FUNCTION_BLOCK fbPiston EXTENDS TcoCore.TcoSequencer

METHOD PROTECTED Main : BOOL


IF Step(10,
TRUE,
'_moveHomeTask') THEN
//-------------------------------------------------------
	IF(_moveHomeTask.Invoke().Done)THEN
		StepCompleteWhen(TRUE);
	END_IF;
//-------------------------------------------------------
END_IF;

IF Step(20,
TRUE,
'_moveWorkTask') THEN
//-------------------------------------------------------
	IF(_moveWorkTask.Invoke().Done)THEN
		StepCompleteWhen(TRUE);
	END_IF;
//-------------------------------------------------------
END_IF;

IF Step(30,
TRUE,
'_moveHomeToggleTask') THEN
//-------------------------------------------------------
	IF(_moveHomeToggleTask.Toggle())THEN
		StepCompleteWhen(TRUE);
	END_IF;
//-------------------------------------------------------
END_IF;

IF Step(40,
TRUE,
'_moveHomeToggleTask') THEN
//-------------------------------------------------------
	IF(_moveHomeToggleTask.Toggle())THEN
		StepCompleteWhen(TRUE);
	END_IF;
//-------------------------------------------------------
END_IF;

IF Step(50,
TRUE,
'_moveHomeMomentaryTask') THEN
//-------------------------------------------------------
	IF(_moveHomeMomentaryTask.On())THEN
		StepCompleteWhen(TRUE);
	END_IF;
//-------------------------------------------------------
END_IF;

IF Step(60,
TRUE,
'_moveHomeMomentaryTask') THEN
//-------------------------------------------------------
	IF(_moveHomeMomentaryTask.Off())THEN
		StepCompleteWhen(TRUE);
	END_IF;
//-------------------------------------------------------
END_IF;
END_METHOD

END_FUNCTION_BLOCK

(* stored: Version 1.1.0.1, ProductVersion 3.1.4024.9
   POU fbPiston: Id {41ce95b1-694a-4bd3-b773-5382b98402d8}, SpecialFunc None
   Method Main: Id {c86ecde6-1911-404c-86d2-9ddbfc0b3cb4} *)
